TYPE EL5152_HWTOPLC_PDOS :
	STRUCT
	
	status												: EL5152_STATUS;	
		{attribute 'hide'}
	_reserved1                                          : UINT;

	CounterValue                              : UDINT; // Current encoder counter value

	END_STRUCT
END_TYPE

(* stored: Version 1.1.0.1
   DUT EL5152_HWTOPLC_PDOS: Id {755519b7-2a5e-408d-a1a6-d3222ca02e2c} *)
